// TIA Portal V16 export
// export: Created 2022-02-04T14:40:19.9325166Z, ExportSetting WithDefaults, DisplayName Totally Integrated Automation Portal, DisplayVersion V16 Update 1, DisplayName TIA Portal Version Control Interface, DisplayVersion V16, DisplayName TIA Portal Openness, DisplayVersion V16, DisplayName SINAMICS Startdrive Advanced, DisplayVersion V16 Update 5, DisplayName SINAMICS Startdrive G130, G150, S120, S150, SINAMICS MV, S210, DisplayVersion V16 Update 5, DisplayName SINAMICS Startdrive G110M, G120, G120C, G120D, G120P, G115D, DisplayVersion V16 Update 5, DisplayName STEP 7 Professional, DisplayVersion V16, DisplayName STEP 7 Safety, DisplayVersion V16, DisplayName WinCC Advanced, DisplayVersion V16, DisplayName SIMATIC Visualization Architect, DisplayVersion V16
DATA_BLOCK "HS"   // DB21
VERSION : 0.1
// stored: AutoNumber true, InstanceOfName FB_HydroStations, InstanceOfType FB
"FB_HydroStations"
   // VAR RETAIN
   //    Upor_resetter : "CyclicSignal";
   //    Movable_side_resetter { S7_SetPoint := 'True'} : "CyclicSignal";
   //    Gasket_Ramp_sync { S7_SetPoint := 'True'} : "CyclicSignal";
   //    DefectDrop_resetter { S7_SetPoint := 'True'} : "CyclicSignal";
   //    Board_Rotator : "FB_IM2x0";
   //    Defect_Drop { S7_SetPoint := 'True'} : "FB_IM2x0";
   //    Upor_Sorting : "FB_IM2x0";
   //    Upor_Defective { S7_SetPoint := 'True'} : "FB_IM2x2";
   //    Gasket_Supplier : "FB_IM2x0";
   //    Gasket_Ramp { S7_SetPoint := 'True'} : "FB_IM2x3";
   //    Gasket_Lodems { S7_SetPoint := 'True'} : "FB_IM2x2";
   //    Forks_Pitcher { S7_SetPoint := 'True'} : "FB_IM2x2";
   //    Movable_Side { S7_SetPoint := 'True'} : "FB_IM2x0";
   //    Upor_PFM { S7_SetPoint := 'True'} : "FB_IM2x0";
   //    M_221_Large_HydroStationDrive { S7_SetPoint := 'True'} : "FB_HySt_Drive_PassValve";
   //    M_337_Small_HydroStationDrive { S7_SetPoint := 'True'} : "FB_HySt_Drive_PassValve";
   // END_VAR
BEGIN
END_DATA_BLOCK
